{attribute 'GeneratedUsingTerminal: BK1150-0000-0016'}
{attribute addProperty BoxType "BK1150-0000-0016"}
{attribute addProperty Id "Term_383_KL1002KL1002_BB38DA8F0"}
{attribute addProperty CRC "2584925327"}
{attribute addProperty Size "0"}
TYPE A_0010_BK1150_0000_0016_9A12D48F EXTENDS BK1150_A2FCADE7 :
STRUCT
	{attribute addProperty Name "Term_383_KL1002"}
	Term_383_KL1002 : KL1002_BB38DA8F;
END_STRUCT
END_TYPE

(* stored: Version 1.2.0.0, ProductVersion 3.1.4024.9
   DUT A_0010_BK1150_0000_0016_9A12D48F: Id {fc979a23-e6fd-406b-8c9a-060dbdd5f785} *)
